{attribute addProperty BoxType "EK1100-0000-0018"}
{attribute addProperty Id "Beckhoff_EL2xxxEK1122Beckhoff_EL2xxxEK1122_8D0C4044162A_0001_EL2002_0000_0000EL2002_39EC201D334.125A_0002_EL2002_0000_0016EL2002_39EC201D334.125A_0003_EL2002_0000_0017EL2002_39EC201D334.125A_0004_EL2002_0000_0018EL2002_39EC201D334.125A_0005_EL2004_0000_0000EL2004_4E3C7537496.125A_0006_EL2004_0000_0016EL2004_4E3C7537496.125A_0007_EL2004_0000_0017EL2004_4E3C7537496.125A_0008_EL2004_0000_0018EL2004_4E3C7537496.125A_0009_EL2008_0000_0016EL2008_A854BE6D8110.125A_0010_EL2008_0000_0017EL2008_A854BE6D8110.125A_0011_EL2008_0000_0018EL2008_A854BE6D8110.125A_0012_EL2014_0000_0016EL2014_B1F56BCC13416.75A_0013_EL2014_0000_0017EL2014_B1F56BCC13416.75A_0014_EL2022_0000_0016EL2022_39EC201D334.125A_0015_EL2022_0000_0017EL2022_39EC201D334.125A_0016_EL2022_0000_0018EL2022_39EC201D334.125A_0017_EL2024_0000_0016EL2024_4E3C7537496.125A_0018_EL2024_0000_0017EL2024_4E3C7537496.125A_0019_EL2024_0000_0018EL2024_4E3C7537496.125A_0020_EL2024_0000_0019EL2024_4E3C7537496.125A_0021_EL2024_0010_0016EL2024_4E3C7537496.125A_0022_EL2024_0010_0017EL2024_4E3C7537496.125A_0023_EL2024_0010_0018EL2024_4E3C7537496.125A_0024_EL2032_0000_0000EL2032_D8352AAE506.25A_0025_EL2032_0000_0016EL2032_D8352AAE506.25A_0026_EL2032_0000_0017EL2032_D8352AAE506.25A_0027_EL2032_0000_0018EL2032_D8352AAE506.25A_0028_EL2034_0000_0016EL2034_14D53AA68210.25A_0029_EL2034_0000_0017EL2034_14D53AA68210.25A_0030_EL2034_0000_0018EL2034_14D53AA68210.25A_0031_EL2042_0000_0016EL2042_39EC201D334.125A_0032_EL2042_0000_0017EL2042_39EC201D334.125A_0033_EL2042_0000_0018EL2042_39EC201D334.125A_0034_EL2044_0000_0016EL2044_B1F56BCC13416.75A_0035_EL2084_0000_0016EL2084_4E3C7537496.125A_0036_EL2084_0000_0017EL2084_4E3C7537496.125A_0037_EL2084_0000_0018EL2084_4E3C7537496.125A_0038_EL2088_0000_0016EL2088_A854BE6D8110.125A_0039_EL2088_0000_0017EL2088_A854BE6D8110.125A_0040_EL2088_0000_0018EL2088_A854BE6D8110.125A_0041_EL2124_0000_0016EL2124_4E3C7537496.125A_0042_EL2124_0000_0017EL2124_4E3C7537496.125A_0043_EL2124_0000_0018EL2124_4E3C7537496.125A_0044_EL2202_0000_0000EL2202_39EC201D334.125A_0045_EL2202_0000_0016EL2202_B7733B6A496.125A_0046_EL2202_0000_0017EL2202_B7733B6A496.125A_0047_EL2202_0000_0018EL2202_B7733B6A496.125A_0048_EL2202_0000_0019EL2202_B7733B6A496.125A_0049_EL2202_0100_0016EL2202_B0EF2F1411314.125A_0050_EL2202_0100_0017EL2202_B0EF2F1411314.125A_0051_EL2202_0100_0018EL2202_B0EF2F1411314.125A_0052_EL2202_0100_0019EL2202_B0EF2F1411314.125A_0053_EL2212_0000_0018EL2212_74FAECA914618.25A_0054_EL2212_0000_0019EL2212_74FAECA914618.25A_0055_EL2212_0000_0020EL2212_1A3ABF1914618.25A_0056_EL2212_0000_0021EL2212_1A3ABF1914618.25A_0057_EL2212_0000_0022EL2212_1A3ABF1914618.25A_0058_EL2212_0000_0023EL2212_1A3ABF1914618.25A_0059_EL2252_0000_0000EL2252_3BE0B4B713717.125A_0060_EL2252_0000_0016EL2252_7A0EDC2E16921.125A_0061_EL2252_0000_0017EL2252_9614143218523.125A_0062_EL2252_0000_0018EL2252_9614143218523.125A_0063_EL2252_0000_0019EL2252_9614143218523.125A_0064_EL2252_0000_0020EL2252_9614143218523.125A_0065_EL2258_0000_0016EL2258_0502BFA15602700.25A_0066_EL2258_0000_0017EL2258_9BBCB8E35546693.25A_0067_EL2262_0000_0000EL2262_D2325A4710513.125A_0068_EL2262_0000_0001EL2262_6FCF2F7B12916.125A_0069_EL2262_0000_0002EL2262_131C31B227334.125A_0070_EL2262_0000_0003EL2262_131C31B227334.125A_0071_EL2262_0000_0004EL2262_E0ACD1AC30638.25A_0072_EL2602_0000_0016EL2602_39EC201D334.125A_0073_EL2602_0000_0017EL2602_39EC201D334.125A_0074_EL2602_0000_0018EL2602_39EC201D334.125A_0075_EL2602_0010_0016EL2602_452236B5425.25A_0076_EL2612_0000_0016EL2612_39EC201D334.125A_0077_EL2612_0000_0017EL2612_39EC201D334.125A_0078_EL2612_0000_0018EL2612_39EC201D334.125A_0079_EL2622_0000_0016EL2622_39EC201D334.125A_0080_EL2622_0000_0017EL2622_39EC201D334.125A_0081_EL2622_0000_0018EL2622_39EC201D334.125A_0082_EL2622_0010_0016EL2622_452236B5425.25A_0083_EL2624_0000_0016EL2624_4E3C7537496.125A_0084_EL2624_0000_0017EL2624_4E3C7537496.125A_0085_EL2624_0000_0018EL2624_4E3C7537496.125A_0086_EL2634_0000_0016EL2634_4E3C7537496.125A_0087_EL2634_0000_0017EL2634_4E3C7537496.125A_0088_EL2642_0000_0016EL2642_1DA2CD0419424.25A_0089_EL2652_0000_0016EL2652_39EC201D334.125A_0090_EL2652_0000_0017EL2652_39EC201D334.125A_0091_EL2652_0000_0018EL2652_39EC201D334.125A_0092_EL2712_0000_0016EL2712_39EC201D334.125A_0093_EL2712_0000_0017EL2712_39EC201D334.125A_0094_EL2722_0000_0016EL2722_39EC201D334.125A_0095_EL2722_0010_0016EL2722_39EC201D334.125A_0096_EL2732_0000_0016EL2732_39EC201D334.125A_0097_EL2784_0000_0016EL2784_4E3C7537496.125A_0098_EL2788_0000_0016EL2788_A854BE6D8110.125A_0099_EL2794_0000_0016EL2794_4E3C7537496.125A_0100_EL2798_0000_0016EL2798_A854BE6D8110.125A_0101_EL2798_0000_0017EL2798_A854BE6D8110.125A_0102_EL2798_0000_0018EL2798_A854BE6D8110.125A_0103_EL2808_0000_0016EL2808_A854BE6D8110.125A_0104_EL2808_0000_0017EL2808_A854BE6D8110.125A_0105_EL2808_0000_0018EL2808_A854BE6D8110.125A_0106_EL2809_0000_0016EL2809_859F43D214518.125A_0107_EL2809_0000_0017EL2809_859F43D214518.125A_0108_EL2809_0000_0018EL2809_859F43D214518.125A_0109_EL2819_0000_0016EL2819_84B65E3F19424.25A_0110_EL2819_0000_0017EL2819_84B65E3F19424.25A_0111_EL2819_0000_0018EL2819_84B65E3F19424.25A_0112_EL2828_0000_0016EL2828_A854BE6D8110.125A_0113_EL2828_0000_0017EL2828_A854BE6D8110.125A_0114_EL2872_0000_0016EL2872_859F43D214518.125A_0115_EL2872_0000_0017EL2872_859F43D214518.125A_0116_EL2872_0000_0018EL2872_859F43D214518.125A_0117_EL2872_0000_0019EL2872_859F43D214518.125A_0118_EL2872_0010_0016EL2872_859F43D214518.125A_0119_EL2872_0010_0017EL2872_859F43D214518.125A_0120_EL2872_0010_0018EL2872_859F43D214518.125A_0121_EL2872_0010_0019EL2872_859F43D214518.125A_0122_EL2878_0005_0016EL2878_3D5C112B9011.25A_0123_EL2889_0000_0016EL2889_859F43D214518.125A_0124_EL2889_0000_0017EL2889_859F43D214518.125A_0125_EL2889_0000_0018EL2889_859F43D214518.125A_0126_ELM2642_0000_0016ELM2642_A0E9379519424.25A_0127_ELM2644_0000_0016ELM2644_154AC0EC22628.25A_0128_ELM2742_0000_0016ELM2742_A0E9379519424.25A_0129_ELM2744_0000_0016ELM2744_154AC0EC22628.25"}
{attribute addProperty CRC "1834027119"}
{attribute addProperty SizeInBites "22803"}
{attribute addProperty SizeInBytes "2850.375"}
TYPE Beckhoff_EL2xxx_6D51086F EXTENDS EK1100_179A0949 :
STRUCT
	{attribute addProperty Name "Beckhoff_EL2xxxEK1122"}
	Beckhoff_EL2xxxEK1122 : Beckhoff_EL2xxxEK1122_8D0C4044;
	{attribute addProperty Name "A_0001_EL2002_0000_0000"}
	A_0001_EL2002_0000_0000 : EL2002_39EC201D;
	{attribute addProperty Name "A_0002_EL2002_0000_0016"}
	A_0002_EL2002_0000_0016 : EL2002_39EC201D;
	{attribute addProperty Name "A_0003_EL2002_0000_0017"}
	A_0003_EL2002_0000_0017 : EL2002_39EC201D;
	{attribute addProperty Name "A_0004_EL2002_0000_0018"}
	A_0004_EL2002_0000_0018 : EL2002_39EC201D;
	{attribute addProperty Name "A_0005_EL2004_0000_0000"}
	A_0005_EL2004_0000_0000 : EL2004_4E3C7537;
	{attribute addProperty Name "A_0006_EL2004_0000_0016"}
	A_0006_EL2004_0000_0016 : EL2004_4E3C7537;
	{attribute addProperty Name "A_0007_EL2004_0000_0017"}
	A_0007_EL2004_0000_0017 : EL2004_4E3C7537;
	{attribute addProperty Name "A_0008_EL2004_0000_0018"}
	A_0008_EL2004_0000_0018 : EL2004_4E3C7537;
	{attribute addProperty Name "A_0009_EL2008_0000_0016"}
	A_0009_EL2008_0000_0016 : EL2008_A854BE6D;
	{attribute addProperty Name "A_0010_EL2008_0000_0017"}
	A_0010_EL2008_0000_0017 : EL2008_A854BE6D;
	{attribute addProperty Name "A_0011_EL2008_0000_0018"}
	A_0011_EL2008_0000_0018 : EL2008_A854BE6D;
	{attribute addProperty Name "A_0012_EL2014_0000_0016"}
	A_0012_EL2014_0000_0016 : EL2014_B1F56BCC;
	{attribute addProperty Name "A_0013_EL2014_0000_0017"}
	A_0013_EL2014_0000_0017 : EL2014_B1F56BCC;
	{attribute addProperty Name "A_0014_EL2022_0000_0016"}
	A_0014_EL2022_0000_0016 : EL2022_39EC201D;
	{attribute addProperty Name "A_0015_EL2022_0000_0017"}
	A_0015_EL2022_0000_0017 : EL2022_39EC201D;
	{attribute addProperty Name "A_0016_EL2022_0000_0018"}
	A_0016_EL2022_0000_0018 : EL2022_39EC201D;
	{attribute addProperty Name "A_0017_EL2024_0000_0016"}
	A_0017_EL2024_0000_0016 : EL2024_4E3C7537;
	{attribute addProperty Name "A_0018_EL2024_0000_0017"}
	A_0018_EL2024_0000_0017 : EL2024_4E3C7537;
	{attribute addProperty Name "A_0019_EL2024_0000_0018"}
	A_0019_EL2024_0000_0018 : EL2024_4E3C7537;
	{attribute addProperty Name "A_0020_EL2024_0000_0019"}
	A_0020_EL2024_0000_0019 : EL2024_4E3C7537;
	{attribute addProperty Name "A_0021_EL2024_0010_0016"}
	A_0021_EL2024_0010_0016 : EL2024_4E3C7537;
	{attribute addProperty Name "A_0022_EL2024_0010_0017"}
	A_0022_EL2024_0010_0017 : EL2024_4E3C7537;
	{attribute addProperty Name "A_0023_EL2024_0010_0018"}
	A_0023_EL2024_0010_0018 : EL2024_4E3C7537;
	{attribute addProperty Name "A_0024_EL2032_0000_0000"}
	A_0024_EL2032_0000_0000 : EL2032_D8352AAE;
	{attribute addProperty Name "A_0025_EL2032_0000_0016"}
	A_0025_EL2032_0000_0016 : EL2032_D8352AAE;
	{attribute addProperty Name "A_0026_EL2032_0000_0017"}
	A_0026_EL2032_0000_0017 : EL2032_D8352AAE;
	{attribute addProperty Name "A_0027_EL2032_0000_0018"}
	A_0027_EL2032_0000_0018 : EL2032_D8352AAE;
	{attribute addProperty Name "A_0028_EL2034_0000_0016"}
	A_0028_EL2034_0000_0016 : EL2034_14D53AA6;
	{attribute addProperty Name "A_0029_EL2034_0000_0017"}
	A_0029_EL2034_0000_0017 : EL2034_14D53AA6;
	{attribute addProperty Name "A_0030_EL2034_0000_0018"}
	A_0030_EL2034_0000_0018 : EL2034_14D53AA6;
	{attribute addProperty Name "A_0031_EL2042_0000_0016"}
	A_0031_EL2042_0000_0016 : EL2042_39EC201D;
	{attribute addProperty Name "A_0032_EL2042_0000_0017"}
	A_0032_EL2042_0000_0017 : EL2042_39EC201D;
	{attribute addProperty Name "A_0033_EL2042_0000_0018"}
	A_0033_EL2042_0000_0018 : EL2042_39EC201D;
	{attribute addProperty Name "A_0034_EL2044_0000_0016"}
	A_0034_EL2044_0000_0016 : EL2044_B1F56BCC;
	{attribute addProperty Name "A_0035_EL2084_0000_0016"}
	A_0035_EL2084_0000_0016 : EL2084_4E3C7537;
	{attribute addProperty Name "A_0036_EL2084_0000_0017"}
	A_0036_EL2084_0000_0017 : EL2084_4E3C7537;
	{attribute addProperty Name "A_0037_EL2084_0000_0018"}
	A_0037_EL2084_0000_0018 : EL2084_4E3C7537;
	{attribute addProperty Name "A_0038_EL2088_0000_0016"}
	A_0038_EL2088_0000_0016 : EL2088_A854BE6D;
	{attribute addProperty Name "A_0039_EL2088_0000_0017"}
	A_0039_EL2088_0000_0017 : EL2088_A854BE6D;
	{attribute addProperty Name "A_0040_EL2088_0000_0018"}
	A_0040_EL2088_0000_0018 : EL2088_A854BE6D;
	{attribute addProperty Name "A_0041_EL2124_0000_0016"}
	A_0041_EL2124_0000_0016 : EL2124_4E3C7537;
	{attribute addProperty Name "A_0042_EL2124_0000_0017"}
	A_0042_EL2124_0000_0017 : EL2124_4E3C7537;
	{attribute addProperty Name "A_0043_EL2124_0000_0018"}
	A_0043_EL2124_0000_0018 : EL2124_4E3C7537;
	{attribute addProperty Name "A_0044_EL2202_0000_0000"}
	A_0044_EL2202_0000_0000 : EL2202_39EC201D;
	{attribute addProperty Name "A_0045_EL2202_0000_0016"}
	A_0045_EL2202_0000_0016 : EL2202_B7733B6A;
	{attribute addProperty Name "A_0046_EL2202_0000_0017"}
	A_0046_EL2202_0000_0017 : EL2202_B7733B6A;
	{attribute addProperty Name "A_0047_EL2202_0000_0018"}
	A_0047_EL2202_0000_0018 : EL2202_B7733B6A;
	{attribute addProperty Name "A_0048_EL2202_0000_0019"}
	A_0048_EL2202_0000_0019 : EL2202_B7733B6A;
	{attribute addProperty Name "A_0049_EL2202_0100_0016"}
	A_0049_EL2202_0100_0016 : EL2202_B0EF2F14;
	{attribute addProperty Name "A_0050_EL2202_0100_0017"}
	A_0050_EL2202_0100_0017 : EL2202_B0EF2F14;
	{attribute addProperty Name "A_0051_EL2202_0100_0018"}
	A_0051_EL2202_0100_0018 : EL2202_B0EF2F14;
	{attribute addProperty Name "A_0052_EL2202_0100_0019"}
	A_0052_EL2202_0100_0019 : EL2202_B0EF2F14;
	{attribute addProperty Name "A_0053_EL2212_0000_0018"}
	A_0053_EL2212_0000_0018 : EL2212_74FAECA9;
	{attribute addProperty Name "A_0054_EL2212_0000_0019"}
	A_0054_EL2212_0000_0019 : EL2212_74FAECA9;
	{attribute addProperty Name "A_0055_EL2212_0000_0020"}
	A_0055_EL2212_0000_0020 : EL2212_1A3ABF19;
	{attribute addProperty Name "A_0056_EL2212_0000_0021"}
	A_0056_EL2212_0000_0021 : EL2212_1A3ABF19;
	{attribute addProperty Name "A_0057_EL2212_0000_0022"}
	A_0057_EL2212_0000_0022 : EL2212_1A3ABF19;
	{attribute addProperty Name "A_0058_EL2212_0000_0023"}
	A_0058_EL2212_0000_0023 : EL2212_1A3ABF19;
	{attribute addProperty Name "A_0059_EL2252_0000_0000"}
	A_0059_EL2252_0000_0000 : EL2252_3BE0B4B7;
	{attribute addProperty Name "A_0060_EL2252_0000_0016"}
	A_0060_EL2252_0000_0016 : EL2252_7A0EDC2E;
	{attribute addProperty Name "A_0061_EL2252_0000_0017"}
	A_0061_EL2252_0000_0017 : EL2252_96141432;
	{attribute addProperty Name "A_0062_EL2252_0000_0018"}
	A_0062_EL2252_0000_0018 : EL2252_96141432;
	{attribute addProperty Name "A_0063_EL2252_0000_0019"}
	A_0063_EL2252_0000_0019 : EL2252_96141432;
	{attribute addProperty Name "A_0064_EL2252_0000_0020"}
	A_0064_EL2252_0000_0020 : EL2252_96141432;
	{attribute addProperty Name "A_0065_EL2258_0000_0016"}
	A_0065_EL2258_0000_0016 : EL2258_0502BFA1;
	{attribute addProperty Name "A_0066_EL2258_0000_0017"}
	A_0066_EL2258_0000_0017 : EL2258_9BBCB8E3;
	{attribute addProperty Name "A_0067_EL2262_0000_0000"}
	A_0067_EL2262_0000_0000 : EL2262_D2325A47;
	{attribute addProperty Name "A_0068_EL2262_0000_0001"}
	A_0068_EL2262_0000_0001 : EL2262_6FCF2F7B;
	{attribute addProperty Name "A_0069_EL2262_0000_0002"}
	A_0069_EL2262_0000_0002 : EL2262_131C31B2;
	{attribute addProperty Name "A_0070_EL2262_0000_0003"}
	A_0070_EL2262_0000_0003 : EL2262_131C31B2;
	{attribute addProperty Name "A_0071_EL2262_0000_0004"}
	A_0071_EL2262_0000_0004 : EL2262_E0ACD1AC;
	{attribute addProperty Name "A_0072_EL2602_0000_0016"}
	A_0072_EL2602_0000_0016 : EL2602_39EC201D;
	{attribute addProperty Name "A_0073_EL2602_0000_0017"}
	A_0073_EL2602_0000_0017 : EL2602_39EC201D;
	{attribute addProperty Name "A_0074_EL2602_0000_0018"}
	A_0074_EL2602_0000_0018 : EL2602_39EC201D;
	{attribute addProperty Name "A_0075_EL2602_0010_0016"}
	A_0075_EL2602_0010_0016 : EL2602_452236B5;
	{attribute addProperty Name "A_0076_EL2612_0000_0016"}
	A_0076_EL2612_0000_0016 : EL2612_39EC201D;
	{attribute addProperty Name "A_0077_EL2612_0000_0017"}
	A_0077_EL2612_0000_0017 : EL2612_39EC201D;
	{attribute addProperty Name "A_0078_EL2612_0000_0018"}
	A_0078_EL2612_0000_0018 : EL2612_39EC201D;
	{attribute addProperty Name "A_0079_EL2622_0000_0016"}
	A_0079_EL2622_0000_0016 : EL2622_39EC201D;
	{attribute addProperty Name "A_0080_EL2622_0000_0017"}
	A_0080_EL2622_0000_0017 : EL2622_39EC201D;
	{attribute addProperty Name "A_0081_EL2622_0000_0018"}
	A_0081_EL2622_0000_0018 : EL2622_39EC201D;
	{attribute addProperty Name "A_0082_EL2622_0010_0016"}
	A_0082_EL2622_0010_0016 : EL2622_452236B5;
	{attribute addProperty Name "A_0083_EL2624_0000_0016"}
	A_0083_EL2624_0000_0016 : EL2624_4E3C7537;
	{attribute addProperty Name "A_0084_EL2624_0000_0017"}
	A_0084_EL2624_0000_0017 : EL2624_4E3C7537;
	{attribute addProperty Name "A_0085_EL2624_0000_0018"}
	A_0085_EL2624_0000_0018 : EL2624_4E3C7537;
	{attribute addProperty Name "A_0086_EL2634_0000_0016"}
	A_0086_EL2634_0000_0016 : EL2634_4E3C7537;
	{attribute addProperty Name "A_0087_EL2634_0000_0017"}
	A_0087_EL2634_0000_0017 : EL2634_4E3C7537;
	{attribute addProperty Name "A_0088_EL2642_0000_0016"}
	A_0088_EL2642_0000_0016 : EL2642_1DA2CD04;
	{attribute addProperty Name "A_0089_EL2652_0000_0016"}
	A_0089_EL2652_0000_0016 : EL2652_39EC201D;
	{attribute addProperty Name "A_0090_EL2652_0000_0017"}
	A_0090_EL2652_0000_0017 : EL2652_39EC201D;
	{attribute addProperty Name "A_0091_EL2652_0000_0018"}
	A_0091_EL2652_0000_0018 : EL2652_39EC201D;
	{attribute addProperty Name "A_0092_EL2712_0000_0016"}
	A_0092_EL2712_0000_0016 : EL2712_39EC201D;
	{attribute addProperty Name "A_0093_EL2712_0000_0017"}
	A_0093_EL2712_0000_0017 : EL2712_39EC201D;
	{attribute addProperty Name "A_0094_EL2722_0000_0016"}
	A_0094_EL2722_0000_0016 : EL2722_39EC201D;
	{attribute addProperty Name "A_0095_EL2722_0010_0016"}
	A_0095_EL2722_0010_0016 : EL2722_39EC201D;
	{attribute addProperty Name "A_0096_EL2732_0000_0016"}
	A_0096_EL2732_0000_0016 : EL2732_39EC201D;
	{attribute addProperty Name "A_0097_EL2784_0000_0016"}
	A_0097_EL2784_0000_0016 : EL2784_4E3C7537;
	{attribute addProperty Name "A_0098_EL2788_0000_0016"}
	A_0098_EL2788_0000_0016 : EL2788_A854BE6D;
	{attribute addProperty Name "A_0099_EL2794_0000_0016"}
	A_0099_EL2794_0000_0016 : EL2794_4E3C7537;
	{attribute addProperty Name "A_0100_EL2798_0000_0016"}
	A_0100_EL2798_0000_0016 : EL2798_A854BE6D;
	{attribute addProperty Name "A_0101_EL2798_0000_0017"}
	A_0101_EL2798_0000_0017 : EL2798_A854BE6D;
	{attribute addProperty Name "A_0102_EL2798_0000_0018"}
	A_0102_EL2798_0000_0018 : EL2798_A854BE6D;
	{attribute addProperty Name "A_0103_EL2808_0000_0016"}
	A_0103_EL2808_0000_0016 : EL2808_A854BE6D;
	{attribute addProperty Name "A_0104_EL2808_0000_0017"}
	A_0104_EL2808_0000_0017 : EL2808_A854BE6D;
	{attribute addProperty Name "A_0105_EL2808_0000_0018"}
	A_0105_EL2808_0000_0018 : EL2808_A854BE6D;
	{attribute addProperty Name "A_0106_EL2809_0000_0016"}
	A_0106_EL2809_0000_0016 : EL2809_859F43D2;
	{attribute addProperty Name "A_0107_EL2809_0000_0017"}
	A_0107_EL2809_0000_0017 : EL2809_859F43D2;
	{attribute addProperty Name "A_0108_EL2809_0000_0018"}
	A_0108_EL2809_0000_0018 : EL2809_859F43D2;
	{attribute addProperty Name "A_0109_EL2819_0000_0016"}
	A_0109_EL2819_0000_0016 : EL2819_84B65E3F;
	{attribute addProperty Name "A_0110_EL2819_0000_0017"}
	A_0110_EL2819_0000_0017 : EL2819_84B65E3F;
	{attribute addProperty Name "A_0111_EL2819_0000_0018"}
	A_0111_EL2819_0000_0018 : EL2819_84B65E3F;
	{attribute addProperty Name "A_0112_EL2828_0000_0016"}
	A_0112_EL2828_0000_0016 : EL2828_A854BE6D;
	{attribute addProperty Name "A_0113_EL2828_0000_0017"}
	A_0113_EL2828_0000_0017 : EL2828_A854BE6D;
	{attribute addProperty Name "A_0114_EL2872_0000_0016"}
	A_0114_EL2872_0000_0016 : EL2872_859F43D2;
	{attribute addProperty Name "A_0115_EL2872_0000_0017"}
	A_0115_EL2872_0000_0017 : EL2872_859F43D2;
	{attribute addProperty Name "A_0116_EL2872_0000_0018"}
	A_0116_EL2872_0000_0018 : EL2872_859F43D2;
	{attribute addProperty Name "A_0117_EL2872_0000_0019"}
	A_0117_EL2872_0000_0019 : EL2872_859F43D2;
	{attribute addProperty Name "A_0118_EL2872_0010_0016"}
	A_0118_EL2872_0010_0016 : EL2872_859F43D2;
	{attribute addProperty Name "A_0119_EL2872_0010_0017"}
	A_0119_EL2872_0010_0017 : EL2872_859F43D2;
	{attribute addProperty Name "A_0120_EL2872_0010_0018"}
	A_0120_EL2872_0010_0018 : EL2872_859F43D2;
	{attribute addProperty Name "A_0121_EL2872_0010_0019"}
	A_0121_EL2872_0010_0019 : EL2872_859F43D2;
	{attribute addProperty Name "A_0122_EL2878_0005_0016"}
	A_0122_EL2878_0005_0016 : EL2878_3D5C112B;
	{attribute addProperty Name "A_0123_EL2889_0000_0016"}
	A_0123_EL2889_0000_0016 : EL2889_859F43D2;
	{attribute addProperty Name "A_0124_EL2889_0000_0017"}
	A_0124_EL2889_0000_0017 : EL2889_859F43D2;
	{attribute addProperty Name "A_0125_EL2889_0000_0018"}
	A_0125_EL2889_0000_0018 : EL2889_859F43D2;
	{attribute addProperty Name "A_0126_ELM2642_0000_0016"}
	A_0126_ELM2642_0000_0016 : ELM2642_A0E93795;
	{attribute addProperty Name "A_0127_ELM2644_0000_0016"}
	A_0127_ELM2644_0000_0016 : ELM2644_154AC0EC;
	{attribute addProperty Name "A_0128_ELM2742_0000_0016"}
	A_0128_ELM2742_0000_0016 : ELM2742_A0E93795;
	{attribute addProperty Name "A_0129_ELM2744_0000_0016"}
	A_0129_ELM2744_0000_0016 : ELM2744_154AC0EC;
END_STRUCT
END_TYPE

(* stored: Version 1.2.0.0, ProductVersion 3.1.4024.9
   DUT Beckhoff_EL2xxx_6D51086F: Id {5f688e51-4a04-48c5-9142-4783c84c9440} *)
